# B&R Automation Studio project LibTeltonikaSms
Automation Studio 4.9

## Configuration Config1

CPU X20CP0484-1, AutomationRuntime 6.0.2, Build 11.3.0, Vc 6.0.0

### Task classes (Cpu.sw)
```
Cyclic#2 (cycle 20000 us, tolerance 20000 us):
  TestProgra <- TestProgram.prg
Binaries: FWRules, TCData, udbdef, BRRole, asfw, iomap, sysconf, arconfig, ashwd, UaCsConfig, ashwac
Libraries: AsBrStr, AsHttp, runtime, TNSms, standard, AsIecCon, astime, AsBrWStr
```

### Hardware
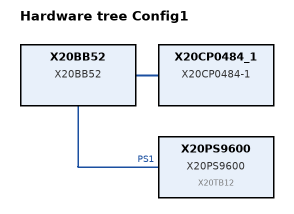
```
X20BB52 : X20BB52 v1.2.0.0
X20CP0484_1 : X20CP0484-1 v1.8.1.0  [SL -> X20BB52.SL1]
  Connector IF2:
    ActivateDevice = 1
    ActivateSnmp = 2
  ConfigurationID = TeltonikaSMS_Config1
  Simulation = 1
  TimerDeviceType = SWIOTIMER
  Cyclic1Duration = 10000
  Cyclic1Tolerance = 10000
  Cyclic1Stack = 16384
  Cyclic2Duration = 20000
  Cyclic2Tolerance = 20000
  Cyclic2Stack = 16384
  Cyclic3Duration = 50000
  Cyclic3Tolerance = 50000
  Cyclic4Duration = 100000
  Cyclic4Tolerance = 100000
  Cyclic5Duration = 200000
  Cyclic5Tolerance = 200000
  Cyclic6Duration = 500000
  Cyclic6Tolerance = 500000
  Cyclic7Duration = 1000000
  Cyclic7Tolerance = 1000000
  Cyclic8Duration = 10000
  Cyclic8Tolerance = 30000000
  FileDevice1
  FileDeviceName1 = USER
  FileDevicePath1 = USER_PATH
  TimeZone = 145
  ActivateWebServer = 1
  ActivateSdm = 1
X20PS9600 : X20PS9600 v1.6.2.0  [PS -> X20BB52.PS1; SS1 -> X20TB12.SS]
X20TB12 : X20TB12 v1.0.0.0
```

## Logical view

Binary libraries used (declarations not repeated): operator, runtime, AsIecCon, astime, AsBrStr, AsHttp, standard, AsBrWStr

### Global.var - Global variables
```iecst
(*PLC Call*)
VAR
	execute : BOOL;
	tnSms0 : teltonikaSms;
END_VAR
(*Router param*)
VAR
	routerIP : STRING[80] := '10.254.254.3';
	routerSmsUser : STRING[80] := 'brplc';
	routerSmsPswd : STRING[80] := 'zkouskaBrPlc1';
END_VAR
(*User data*)
VAR
	ReqType : teltonikaReqType_e := teltonikaReqType_SendMsg;
	EnableData : BOOL := TRUE;
	SimPin : STRING[5] := '0000';
	TelNumber : STRING[20] := '00420123456789';
	Group : STRING[40];
	MsgText : STRING[255] := 'Test SMS - response on another channel';
	MsgId : UDINT := 1;
END_VAR
(*test var*)
VAR
	parsedSmsCount : INT;
	testSmsRead : STRING[2000] := 'Index: 3$nDate: Wed Nov 6 13:32:33 2024$nSender: +420123456789$nText: Stačí?$nStatus: read$n------------------------------$nIndex: 2$nDate: Wed Nov  6 13:32:28 2024$nSender: +420123456789$nText: Blllllll$nStatus: read$n------------------------------$nIndex: 1$nDate: Wed Nov  6 13:32:19 2024$nSender: +420123456789$nText: Hou hej hou hej$nStatus: read$n------------------------------$nIndex: 0$nDate: Wed Nov  6 13:32:00 2024$nSender: +420123456789$nText: Hej hou hej hou$nStatus: read$n------------------------------';
	parsedSms : ARRAY[0..9] OF teltonikaSms_t;
	enableParse : BOOL;
END_VAR
```


### Program Logical/TestProgram (IEC)

#### Main.st
```iecst
PROGRAM _INIT

END_PROGRAM

PROGRAM _CYCLIC
	tnSms0.pRouterAddress := ADR(routerIP);
	tnSms0.pUsername := ADR(routerSmsUser);
	tnSms0.pPassword := ADR(routerSmsPswd);

	tnSms0.requestType := ReqType;
	tnSms0.uEnableData := EnableData;
	tnSms0.upSimPin := ADR(SimPin);
	tnSms0.uMsgId := MsgId;
	tnSms0.upNumber := ADR(TelNumber);
	tnSms0.upGroup := ADR(Group);
	tnSms0.upMsgText := ADR(MsgText);

	tnSms0(enable := TRUE, execute := execute);

	IF enableParse THEN
		enableParse := FALSE;
		parsedSmsCount := teltonikaParseSms(ADR(testSmsRead), SIZEOF(testSmsRead), ADR(parsedSms), SIZEOF(parsedSms)/SIZEOF(teltonikaSms_t));
	END_IF;

END_PROGRAM
```

### Library Logical/TNSms (IEC, version 0.0.1) - Teltonika Network routers SMS sender.
Depends on: AsBrStr, AsHttp, standard

#### Types.typ - Exported data types
```iecst
TYPE
	teltonikaSms_t : 	STRUCT
		index : USINT;
		date : STRING[30];
		sender : STRING[20];
		text : STRING[255];
		status : BOOL;
	END_STRUCT;
END_TYPE

(*Insert your comment here.*)

TYPE
	teltonikaReqType_e :
		(
		teltonikaReqType_EnMobileData,
		teltonikaReqType_SetSimPin,
		teltonikaReqType_ViewMsgList,
		teltonikaReqType_ReadMsg,
		teltonikaReqType_SendMsg,
		teltonikaReqType_SendMsgGroup,
		teltonikaReqType_ViewMsgTotal,
		teltonikaReqType_DeleteMsg
		);
	teltonikaSmsStatus_e :
		(
		teltonikaSmsStatus_NotEnabled,
		teltonikaSmsStatus_Wait,
		teltonikaSmsStatus_Busy,
		teltonikaSmsStatus_Error,
		teltonikaSmsStatus_Ok
		);
END_TYPE

(*Internal automation states*)

TYPE
	tnIntState_e :
		(
		tnIntState_Wait,
		tnIntState_EncodeMsgText,
		tnIntState_CreateReq,
		tnIntState_SendReq,
		tnIntState_WaitForResponse,
		tnIntState_DecodeResponse,
		tnIntState_ParseResponse
		);
END_TYPE
```

#### TNSms.fun - Exported functions and function blocks
```iecst
FUNCTION_BLOCK teltonikaSms
	VAR_INPUT
		enable : BOOL := FALSE; (*Enable block*)
		pRouterAddress : UDINT; (*ADR to string of IP address or DNS name*)
		pUsername : UDINT; (*ADR to string with username*)
		pPassword : UDINT; (*ADR to string with password*)
		requestType : teltonikaReqType_e := teltonikaReqType_ViewMsgTotal; (*Requst type*)
		execute : BOOL := FALSE; (*Execute the command*)
		uEnableData : BOOL := TRUE; (*User - Enable/disable data*)
		upSimPin : UDINT; (*User - ADR of Sim pin to change as string*)
		uMsgId : UDINT; (*User - ID of message to Read or Delete*)
		upNumber : UDINT; (*User - Tel. number of receiver, must be like 0037012345678 (00 + country code + tel. number)*)
		upGroup : UDINT; (*User - group of receivers*)
		upMsgText : UDINT; (*User - ADR of message text*)
	END_VAR
	VAR_OUTPUT
		status : teltonikaSmsStatus_e := (0); (*State of executing. The error or Ok will be for execute state*)
		uMsgCount : INT; (*UserOut - total messages*)
		parsedSms : ARRAY[0..9] OF teltonikaSms_t;
	END_VAR
	VAR
		reExecute : R_TRIG; (*Rise edge for execute*)
		internalState : tnIntState_e; (*Internal state of FUB*)
		requestTypeInternal : teltonikaReqType_e := teltonikaReqType_ViewMsgTotal; (*Requst type*)
		msgTextEncodeUrl : httpEncodeUrl; (*Encoder for URL - change space to %20,...*)
		msgTextEncoded : STRING[3000]; (*It's 1-3 times longer than original*)
		request : STRING[3100]; (*Raw request*)
		requestNxtAddr : UDINT; (*Next address for creating request*)
		reqMsgIdStr : STRING[20]; (*String of message index for creating request*)
		routerSendReq : BOOL; (*Send request to router*)
		routerHttpClient : httpClient;
		routerHttpStatistic : httpStatistics_t;
		routerHttpReqHeader : httpRequestHeader_t;
		routerHttpRespHeader : httpResponseHeader_t;
		routerResponse : STRING[2000]; (*RAW router response*)
		resrponseDecoder : httpUtf8ToString; (*Response decoder from UTF-8 to STRING*)
		decodedResponse : STRING[2000]; (*Decoded router response*)
	END_VAR
END_FUNCTION_BLOCK

FUNCTION teltonikaParseSms : INT
	VAR_INPUT
		pIn : UDINT; (*ADR of input string received from router*)
		sizeIn : UDINT; (*max size of input*)
		pOut : UDINT; (*ADR for output buffer [teltonikaSms_t]*)
		sizeOut : UDINT; (*Array size of output buffer*)
	END_VAR
	VAR
		tmpMem : teltonikaSms_t;
		i : UDINT; (*actual buffer*)
		nextAdrRead : UDINT;
		tmpStrParse : STRING[30];
		tmpStrName : STRING[20];
	END_VAR
END_FUNCTION

FUNCTION tnExtractVal : UDINT
	VAR_INPUT
		pIn : UDINT;
		sizeIn : UDINT;
		pName : UDINT;
		sizeName : UDINT;
		pVal : UDINT;
		sizeVal : UDINT;
	END_VAR
	VAR
		iLen : UDINT;
		nextAddr : UDINT;
		tmpAddr : UDINT;
		actualChar : REFERENCE TO USINT;
	END_VAR
END_FUNCTION

FUNCTION tnFindEndOrLf : UDINT
	VAR_INPUT
		pIn : UDINT;
		sizeIn : UDINT;
	END_VAR
	VAR
		i : UDINT;
		tmpAddr : UDINT;
		actualChar : REFERENCE TO USINT;
	END_VAR
END_FUNCTION
```

#### telttonikaSms.st
```iecst
(* Get spot price of energy from OTE *)
FUNCTION_BLOCK teltonikaSms
	IF NOT enable THEN
		status := teltonikaSmsStatus_NotEnabled;
		RETURN;
	END_IF;

	reExecute(CLK := execute);

	CASE internalState OF
		tnIntState_Wait:
			IF reExecute.Q THEN
				requestTypeInternal := requestType;
				status := teltonikaSmsStatus_Busy;
				internalState := tnIntState_EncodeMsgText;
			END_IF;
			IF NOT execute THEN
				status := teltonikaSmsStatus_Wait;
			END_IF;

		tnIntState_EncodeMsgText:
			internalState := tnIntState_CreateReq;
			IF requestTypeInternal = teltonikaReqType_SendMsg OR requestTypeInternal = teltonikaReqType_SendMsgGroup THEN
				msgTextEncodeUrl(enable := TRUE, pSrc := upMsgText, pDest := ADR(msgTextEncoded), destSize := SIZEOF(msgTextEncoded));
				IF msgTextEncodeUrl.status <> ERR_OK THEN
					internalState := tnIntState_Wait;
					status := teltonikaSmsStatus_Error;
				END_IF;
			END_IF;

		tnIntState_CreateReq:
			request := '';
			requestNxtAddr := ADR(request);
			internalState := tnIntState_SendReq;
			CASE requestTypeInternal OF
				teltonikaReqType_EnMobileData:// /cgi-bin/mobile_date?username=user1&password=user_pass&value=on/off
					requestNxtAddr := brsstrcpy(requestNxtAddr, ADR('/cgi-bin/mobile_date?username='));
					requestNxtAddr := brsstrcpy(requestNxtAddr, pUsername);
					requestNxtAddr := brsstrcpy(requestNxtAddr, ADR('&password='));
					requestNxtAddr := brsstrcpy(requestNxtAddr, pPassword);
					IF uEnableData THEN
						requestNxtAddr := brsstrcpy(requestNxtAddr, ADR('&value=on'));
					ELSE
						requestNxtAddr := brsstrcpy(requestNxtAddr, ADR('&value=off'));
					END_IF;
				teltonikaReqType_SetSimPin:// /cgi-bin/mobile_sim_pin?username=user1&password=user_pass&pin=0000
					requestNxtAddr := brsstrcpy(requestNxtAddr, ADR('/cgi-bin/mobile_sim_pin?username='));
					requestNxtAddr := brsstrcpy(requestNxtAddr, pUsername);
					requestNxtAddr := brsstrcpy(requestNxtAddr, ADR('&password='));
					requestNxtAddr := brsstrcpy(requestNxtAddr, pPassword);
					requestNxtAddr := brsstrcpy(requestNxtAddr, ADR('&pin='));
					requestNxtAddr := brsstrcpy(requestNxtAddr, upSimPin);
				teltonikaReqType_ViewMsgList:// /cgi-bin/sms_list?username=user1&password=user_pass
					requestNxtAddr := brsstrcpy(requestNxtAddr, ADR('/cgi-bin/sms_list?username='));
					requestNxtAddr := brsstrcpy(requestNxtAddr, pUsername);
					requestNxtAddr := brsstrcpy(requestNxtAddr, ADR('&password='));
					requestNxtAddr := brsstrcpy(requestNxtAddr, pPassword);
				teltonikaReqType_ReadMsg:// /cgi-bin/sms_read?username=user1&password=user_pass&number=1
					requestNxtAddr := brsstrcpy(requestNxtAddr, ADR('/cgi-bin/sms_read?username='));
					requestNxtAddr := brsstrcpy(requestNxtAddr, pUsername);
					requestNxtAddr := brsstrcpy(requestNxtAddr, ADR('&password='));
					requestNxtAddr := brsstrcpy(requestNxtAddr, pPassword);
					requestNxtAddr := brsstrcpy(requestNxtAddr, ADR('&number='));
					brsitoa(uMsgId, ADR(reqMsgIdStr));
					requestNxtAddr := brsstrcpy(requestNxtAddr, ADR(reqMsgIdStr));
				teltonikaReqType_SendMsg:// /cgi-bin/sms_send?username=user1&password=user_pass&number=0037060000001&text=testmessage
					requestNxtAddr := brsstrcpy(requestNxtAddr, ADR('/cgi-bin/sms_send?username='));
					requestNxtAddr := brsstrcpy(requestNxtAddr, pUsername);
					requestNxtAddr := brsstrcpy(requestNxtAddr, ADR('&password='));
					requestNxtAddr := brsstrcpy(requestNxtAddr, pPassword);
					requestNxtAddr := brsstrcpy(requestNxtAddr, ADR('&number='));
					requestNxtAddr := brsstrcpy(requestNxtAddr, upNumber);
					requestNxtAddr := brsstrcpy(requestNxtAddr, ADR('&text='));
					requestNxtAddr := brsstrcpy(requestNxtAddr, ADR(msgTextEncoded));
				teltonikaReqType_SendMsgGroup:// /cgi-bin/sms_send?username=user1&password=user_pass&group=group_name&text=testmessage
					requestNxtAddr := brsstrcpy(requestNxtAddr, ADR('/cgi-bin/sms_send?username='));
					requestNxtAddr := brsstrcpy(requestNxtAddr, pUsername);
					requestNxtAddr := brsstrcpy(requestNxtAddr, ADR('&password='));
					requestNxtAddr := brsstrcpy(requestNxtAddr, pPassword);
					requestNxtAddr := brsstrcpy(requestNxtAddr, ADR('&group='));
					requestNxtAddr := brsstrcpy(requestNxtAddr, upGroup);
					requestNxtAddr := brsstrcpy(requestNxtAddr, ADR('&text='));
					requestNxtAddr := brsstrcpy(requestNxtAddr, ADR(msgTextEncoded));
				teltonikaReqType_ViewMsgTotal:// /cgi-bin/sms_total?username=user1&password=user_pass
					requestNxtAddr := brsstrcpy(requestNxtAddr, ADR('/cgi-bin/sms_total?username='));
					requestNxtAddr := brsstrcpy(requestNxtAddr, pUsername);
					requestNxtAddr := brsstrcpy(requestNxtAddr, ADR('&password='));
					requestNxtAddr := brsstrcpy(requestNxtAddr, pPassword);
				teltonikaReqType_DeleteMsg:// /cgi-bin/sms_delete?username=user1&password=user_pass&number=1
					requestNxtAddr := brsstrcpy(requestNxtAddr, ADR('/cgi-bin/sms_delete?username='));
					requestNxtAddr := brsstrcpy(requestNxtAddr, pUsername);
					requestNxtAddr := brsstrcpy(requestNxtAddr, ADR('&password='));
					requestNxtAddr := brsstrcpy(requestNxtAddr, pPassword);
					requestNxtAddr := brsstrcpy(requestNxtAddr, ADR('&number='));
					brsitoa(uMsgId, ADR(reqMsgIdStr));
					requestNxtAddr := brsstrcpy(requestNxtAddr, ADR(reqMsgIdStr));
				ELSE
					internalState := tnIntState_Wait;
					status := teltonikaSmsStatus_Error;
			END_CASE;

		tnIntState_SendReq:
			routerSendReq := TRUE;
			internalState := tnIntState_WaitForResponse;

		tnIntState_WaitForResponse:
			IF DiffDT(routerHttpStatistic.timeOfLastResponse, routerHttpStatistic.timeOfLastRequest) <> 16#FFFFFFFF THEN
				IF (routerHttpClient.status = 0) THEN
					routerSendReq := FALSE;
					IF (routerHttpClient.httpStatus = 200) THEN //Ok
						internalState := tnIntState_DecodeResponse;
					ELSIF routerHttpClient.httpStatus <> 200 THEN //Server error - 400, 404,..
						internalState := tnIntState_Wait;
						status := teltonikaSmsStatus_Error;
					END_IF;
				END_IF;
			END_IF;

		tnIntState_DecodeResponse:
			resrponseDecoder(enable := TRUE, pSrc := ADR(routerResponse), pDest := ADR(decodedResponse), destSize := SIZEOF(decodedResponse), pMappingTable := 0);
			IF resrponseDecoder.status = ERR_OK THEN
				internalState := tnIntState_ParseResponse;
			ELSE
				internalState := tnIntState_Wait;
				status := teltonikaSmsStatus_Error;
			END_IF;

		tnIntState_ParseResponse:
			CASE requestTypeInternal OF
				teltonikaReqType_EnMobileData:

				teltonikaReqType_SetSimPin:

				teltonikaReqType_ViewMsgList:
					uMsgCount := teltonikaParseSms(ADR(routerResponse), SIZEOF(routerResponse), ADR(parsedSms), SIZEOF(parsedSms)/SIZEOF(teltonikaSms_t));

				teltonikaReqType_ReadMsg:
					uMsgCount := teltonikaParseSms(ADR(routerResponse), SIZEOF(routerResponse), ADR(parsedSms), SIZEOF(parsedSms)/SIZEOF(teltonikaSms_t));

				teltonikaReqType_SendMsg:

				teltonikaReqType_SendMsgGroup:

				teltonikaReqType_ViewMsgTotal:

				teltonikaReqType_DeleteMsg:

				ELSE
					internalState := tnIntState_Wait;
					status := teltonikaSmsStatus_Error;
			END_CASE;

			internalState := tnIntState_Wait;
			status := teltonikaSmsStatus_Ok;

		ELSE
			internalState := tnIntState_Wait;
	END_CASE;

	routerHttpClient(enable := TRUE, send := routerSendReq, abort := FALSE, option := httpOPTION_HTTP_11, pHost := pRouterAddress, hostPort := 80, method := httpMETHOD_GET, pUri := ADR(request), pResponseHeader := ADR(routerHttpRespHeader), pResponseData := ADR(routerResponse), responseDataSize := SIZEOF(routerResponse), pStatistics := ADR(routerHttpStatistic), pStruct := 0);

END_FUNCTION_BLOCK

//parse received SMS
FUNCTION teltonikaParseSms
	//Check inputs
	IF sizeIn = 0 OR sizeOut = 0 OR pIn = 0 OR pOut = 0 THEN
		teltonikaParseSms := -1;
		RETURN;
	END_IF;

	teltonikaParseSms := 0;
	brsmemset(pOut, 0, sizeOut * SIZEOF(teltonikaSms_t));//clear output buffer
	nextAdrRead := pIn;

	FOR i := 0 TO sizeOut BY 1 DO
		brsmemset(ADR(tmpMem), 0, SIZEOF(tmpMem));//clear temp data buffer
		//index
		nextAdrRead := tnExtractVal(nextAdrRead, (pIn + sizeIn) - nextAdrRead, ADR(tmpStrName), SIZEOF(tmpStrName), ADR(tmpStrParse), SIZEOF(tmpStrParse));
		IF nextAdrRead = 0 THEN
			teltonikaParseSms := -1;
		END_IF;
		tmpMem.index := DINT_TO_USINT(brsatoi(ADR(tmpStrParse)));

		//date
		nextAdrRead := tnExtractVal(nextAdrRead, (pIn + sizeIn) - nextAdrRead, ADR(tmpStrName), SIZEOF(tmpStrName), ADR(tmpMem.date), SIZEOF(tmpMem.date));
		IF nextAdrRead = 0 THEN
			teltonikaParseSms := -1;
		END_IF;
		//tmpMem.date := STRING_TO_DT(tmpStrParse);

		//sender
		nextAdrRead := tnExtractVal(nextAdrRead, (pIn + sizeIn) - nextAdrRead, ADR(tmpStrName), SIZEOF(tmpStrName), ADR(tmpMem.sender), SIZEOF(tmpMem.sender));
		IF nextAdrRead = 0 THEN
			teltonikaParseSms := -1;
		END_IF;

		//text
		nextAdrRead := tnExtractVal(nextAdrRead, (pIn + sizeIn) - nextAdrRead, ADR(tmpStrName), SIZEOF(tmpStrName), ADR(tmpMem.text), SIZEOF(tmpMem.text));
		IF nextAdrRead = 0 THEN
			teltonikaParseSms := -1;
		END_IF;

		//status
		nextAdrRead := tnExtractVal(nextAdrRead, (pIn + sizeIn) - nextAdrRead, ADR(tmpStrName), SIZEOF(tmpStrName), ADR(tmpStrParse), SIZEOF(tmpStrParse));
		IF nextAdrRead = 0 THEN
			teltonikaParseSms := -1;
		END_IF;
		tmpMem.status := brsmemcmp(ADR(tmpStrParse), ADR('read'), 4) = 0;

		brsmemcpy(pOut + i * SIZEOF(teltonikaSms_t), ADR(tmpMem), SIZEOF(teltonikaSms_t));//copy data to buffer

		nextAdrRead := tnFindEndOrLf(nextAdrRead, (pIn + sizeIn) - nextAdrRead);
		IF nextAdrRead = 0 THEN
			teltonikaParseSms := UDINT_TO_INT(i);
			RETURN;
		END_IF;

	END_FOR;
END_FUNCTION

FUNCTION tnExtractVal
	IF pIn = 0 OR sizeIn = 0 OR pName = 0 OR sizeName = 0 OR pVal = 0 OR sizeVal = 0 THEN
		tnExtractVal := 0;
		RETURN;
	END_IF;
	brsmemset(pName, 0, sizeName);
	brsmemset(pVal, 0, sizeVal);

	nextAddr := pIn;
	tmpAddr := pIn;

	iLen := 0;

	//Name
	WHILE tmpAddr < (pIn + sizeIn) DO
		actualChar ACCESS tmpAddr;
		IF actualChar = 58 THEN
			EXIT;
		END_IF;
		tmpAddr := tmpAddr + 1;
		iLen := iLen + 1;
	END_WHILE;
	IF iLen >= sizeName THEN
		tnExtractVal := 0;
		RETURN;
	END_IF;
	brsmemcpy(pName, nextAddr, iLen);
	//
	nextAddr := nextAddr + iLen + 2;
	tmpAddr := tmpAddr + 2;
	iLen := 0;
	//Value
	WHILE tmpAddr < (pIn + sizeIn) DO
		actualChar ACCESS tmpAddr;
		IF actualChar = 10 THEN
			EXIT;
		END_IF;
		tmpAddr := tmpAddr + 1;
		iLen := iLen + 1;
	END_WHILE;
	IF iLen >= sizeVal THEN
		tnExtractVal := 0;
		RETURN;
	END_IF;
	brsmemcpy(pVal, nextAddr, iLen);

	tnExtractVal := nextAddr + iLen + 1;
END_FUNCTION

FUNCTION tnFindEndOrLf
	//Input check
	IF pIn = 0 OR sizeIn = 0 THEN
		tnFindEndOrLf := 0;
		RETURN;
	END_IF;
	//find end char
	tmpAddr := pIn;
	FOR i := 2 TO sizeIn BY 1 DO
		actualChar ACCESS tmpAddr;
		tmpAddr := tmpAddr + 1;
		IF actualChar = 10 OR actualChar = 0 THEN
			tnFindEndOrLf := tmpAddr;
			RETURN;
		END_IF;
	END_FOR;
	tnFindEndOrLf := 0;
END_FUNCTION
```

Listed in the project but not available here: Logical/Global.typ, Logical/TNSms/Constants.var
